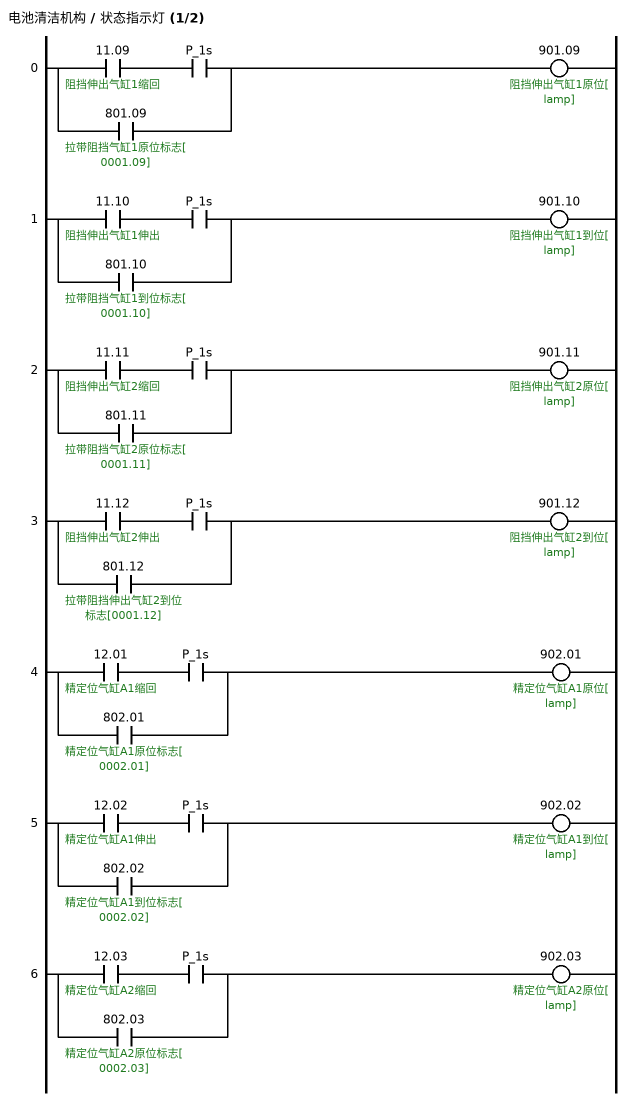
; [picture p72: 电池清洁机构 / 状态指示灯, rungs 0-6]
; rung 0
LD 11.09  ; 阻挡伸出气缸1缩回
AND P_1s
OR 801.09  ; 拉带阻挡气缸1原位标志[0001.09]
OUT 901.09  ; 阻挡伸出气缸1原位[lamp]
; rung 1
LD 11.10  ; 阻挡伸出气缸1伸出
AND P_1s
OR 801.10  ; 拉带阻挡气缸1到位标志[0001.10]
OUT 901.10  ; 阻挡伸出气缸1到位[lamp]
; rung 2
LD 11.11  ; 阻挡伸出气缸2缩回
AND P_1s
OR 801.11  ; 拉带阻挡气缸2原位标志[0001.11]
OUT 901.11  ; 阻挡伸出气缸2原位[lamp]
; rung 3
LD 11.12  ; 阻挡伸出气缸2伸出
AND P_1s
OR 801.12  ; 拉带阻挡伸出气缸2到位标志[0001.12]
OUT 901.12  ; 阻挡伸出气缸2到位[lamp]
; rung 4
LD 12.01  ; 精定位气缸A1缩回
AND P_1s
OR 802.01  ; 精定位气缸A1原位标志[0002.01]
OUT 902.01  ; 精定位气缸A1原位[lamp]
; rung 5
LD 12.02  ; 精定位气缸A1伸出
AND P_1s
OR 802.02  ; 精定位气缸A1到位标志[0002.02]
OUT 902.02  ; 精定位气缸A1到位[lamp]
; rung 6
LD 12.03  ; 精定位气缸A2缩回
AND P_1s
OR 802.03  ; 精定位气缸A2原位标志[0002.03]
OUT 902.03  ; 精定位气缸A2原位[lamp]

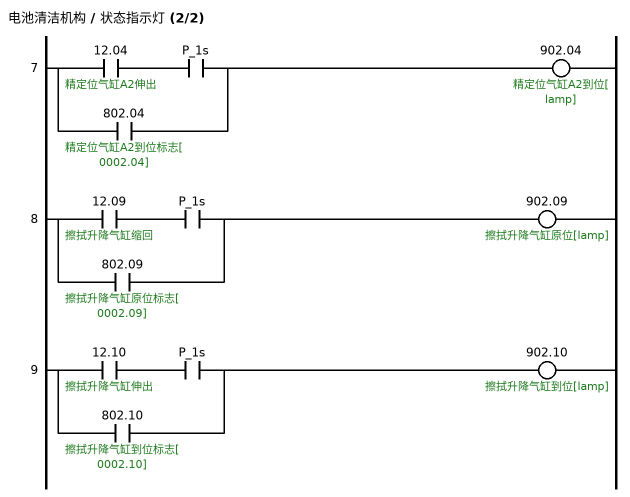
; rung 7
LD 12.04  ; 精定位气缸A2伸出
AND P_1s
OR 802.04  ; 精定位气缸A2到位标志[0002.04]
OUT 902.04  ; 精定位气缸A2到位[lamp]
; rung 8
LD 12.09  ; 擦拭升降气缸缩回
AND P_1s
OR 802.09  ; 擦拭升降气缸原位标志[0002.09]
OUT 902.09  ; 擦拭升降气缸原位[lamp]
; rung 9
LD 12.10  ; 擦拭升降气缸伸出
AND P_1s
OR 802.10  ; 擦拭升降气缸到位标志[0002.10]
OUT 902.10  ; 擦拭升降气缸到位[lamp]

### Section 输出程序

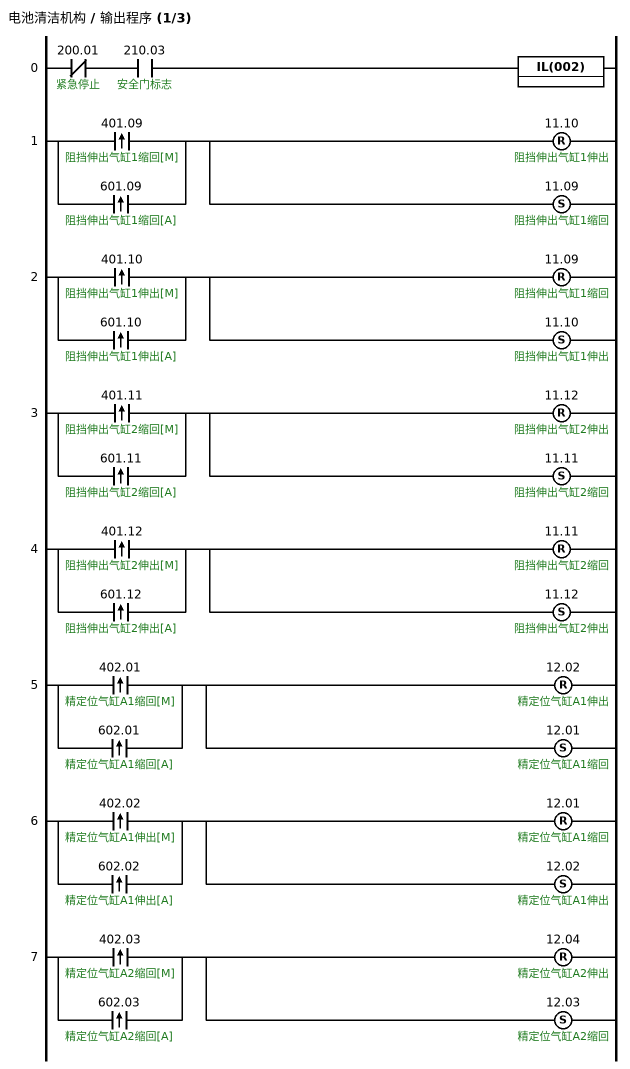
; rung 0
LDNOT 200.01  ; 紧急停止
AND 210.03  ; 安全门标志
IL(002)
; rung 1
@LD 401.09  ; 阻挡伸出气缸1缩回[M]
@OR 601.09  ; 阻挡伸出气缸1缩回[A]
RSET 11.10  ; 阻挡伸出气缸1伸出
SET 11.09  ; 阻挡伸出气缸1缩回
; rung 2
@LD 401.10  ; 阻挡伸出气缸1伸出[M]
@OR 601.10  ; 阻挡伸出气缸1伸出[A]
RSET 11.09  ; 阻挡伸出气缸1缩回
SET 11.10  ; 阻挡伸出气缸1伸出
; rung 3
@LD 401.11  ; 阻挡伸出气缸2缩回[M]
@OR 601.11  ; 阻挡伸出气缸2缩回[A]
RSET 11.12  ; 阻挡伸出气缸2伸出
SET 11.11  ; 阻挡伸出气缸2缩回
; rung 4
@LD 401.12  ; 阻挡伸出气缸2伸出[M]
@OR 601.12  ; 阻挡伸出气缸2伸出[A]
RSET 11.11  ; 阻挡伸出气缸2缩回
SET 11.12  ; 阻挡伸出气缸2伸出
; rung 5
@LD 402.01  ; 精定位气缸A1缩回[M]
@OR 602.01  ; 精定位气缸A1缩回[A]
RSET 12.02  ; 精定位气缸A1伸出
SET 12.01  ; 精定位气缸A1缩回
; rung 6
@LD 402.02  ; 精定位气缸A1伸出[M]
@OR 602.02  ; 精定位气缸A1伸出[A]
RSET 12.01  ; 精定位气缸A1缩回
SET 12.02  ; 精定位气缸A1伸出
; rung 7
@LD 402.03  ; 精定位气缸A2缩回[M]
@OR 602.03  ; 精定位气缸A2缩回[A]
RSET 12.04  ; 精定位气缸A2伸出
SET 12.03  ; 精定位气缸A2缩回

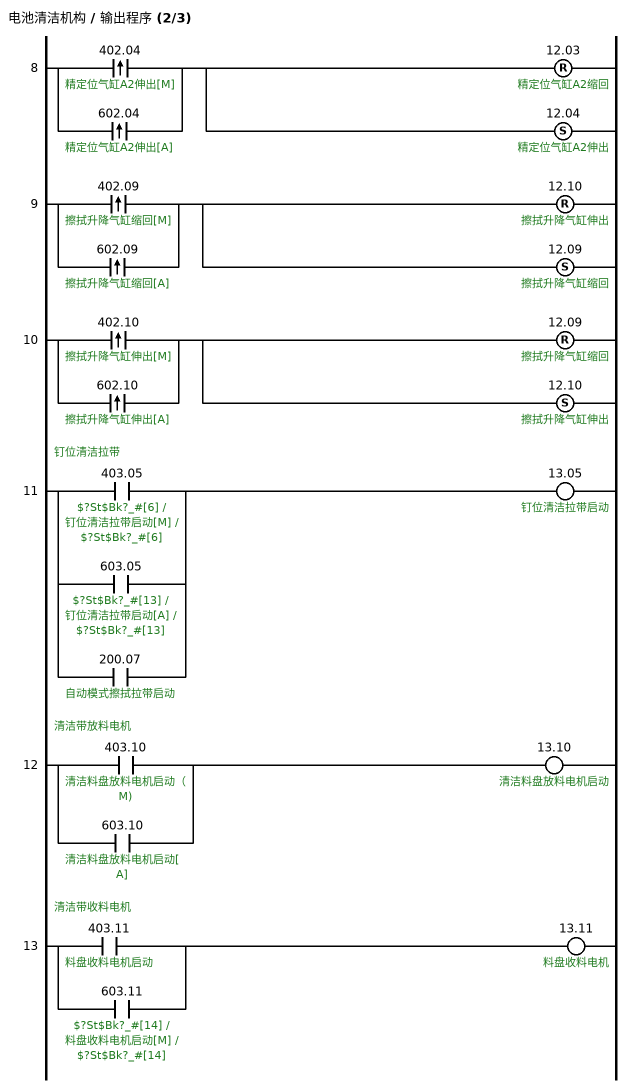
; rung 8
@LD 402.04  ; 精定位气缸A2伸出[M]
@OR 602.04  ; 精定位气缸A2伸出[A]
RSET 12.03  ; 精定位气缸A2缩回
SET 12.04  ; 精定位气缸A2伸出
; rung 9
@LD 402.09  ; 擦拭升降气缸缩回[M]
@OR 602.09  ; 擦拭升降气缸缩回[A]
RSET 12.10  ; 擦拭升降气缸伸出
SET 12.09  ; 擦拭升降气缸缩回
; rung 10
@LD 402.10  ; 擦拭升降气缸伸出[M]
@OR 602.10  ; 擦拭升降气缸伸出[A]
RSET 12.09  ; 擦拭升降气缸缩回
SET 12.10  ; 擦拭升降气缸伸出
; rung 11: 钉位清洁拉带
LD 403.05  ; $?St$Bk?_#[6] / 钉位清洁拉带启动[M] / $?St$Bk?_#[6]
OR 603.05  ; $?St$Bk?_#[13] / 钉位清洁拉带启动[A] / $?St$Bk?_#[13]
OR 200.07  ; 自动模式擦拭拉带启动
OUT 13.05  ; 钉位清洁拉带启动
; rung 12: 清洁带放料电机
LD 403.10  ; 清洁料盘放料电机启动（M)
OR 603.10  ; 清洁料盘放料电机启动[A]
OUT 13.10  ; 清洁料盘放料电机启动
; rung 13: 清洁带收料电机
LD 403.11  ; 料盘收料电机启动
OR 603.11  ; $?St$Bk?_#[14] / 料盘收料电机启动[M] / $?St$Bk?_#[14]
OUT 13.11  ; 料盘收料电机

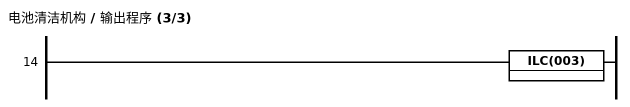
; rung 14
ILC(003)

### Section 擦拭步进电机参数

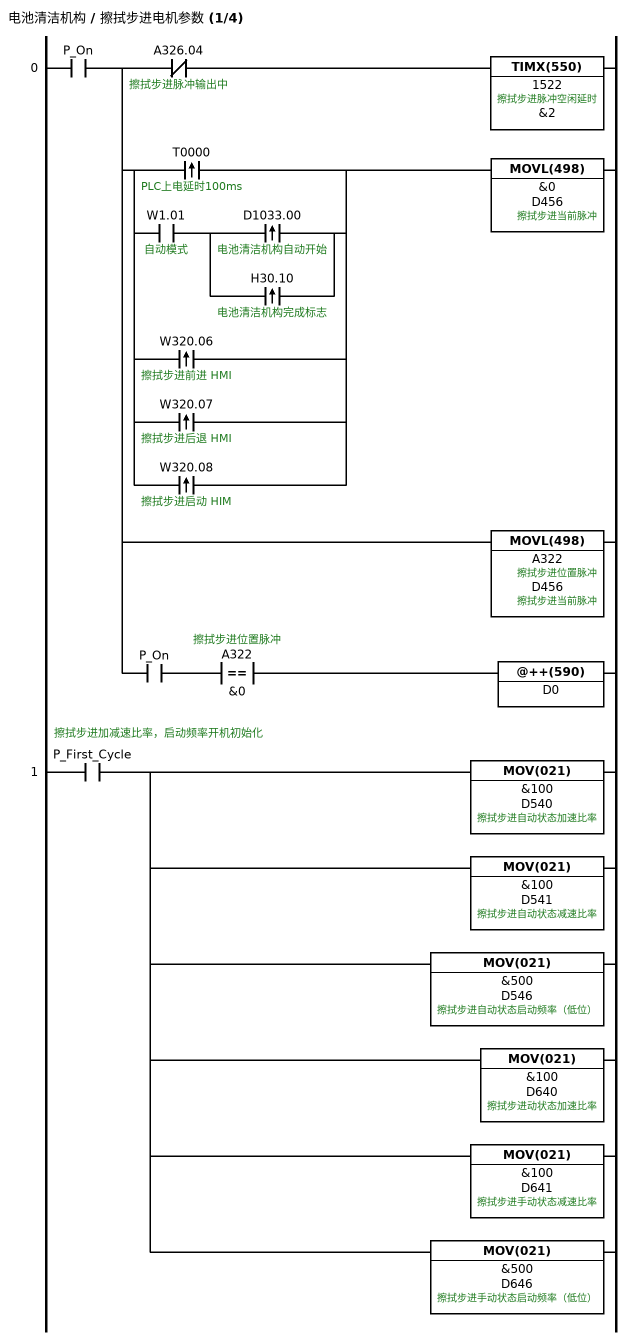
; rung 0
LD P_On
OUT TR0
ANDNOT A326.04  ; 擦拭步进脉冲输出中
TIMX(550) 1522 &2  ; 擦拭步进脉冲空闲延时
LD TR0
@LD T0000  ; PLC上电延时100ms
LD W1.01  ; 自动模式
@LD D1033.00  ; 电池清洁机构自动开始
@OR H30.10  ; 电池清洁机构完成标志
ANDLD
ORLD
@OR W320.06  ; 擦拭步进前进 HMI
@OR W320.07  ; 擦拭步进后退 HMI
@OR W320.08  ; 擦拭步进启动 HIM
ANDLD
MOVL(498) &0 D456  ; 擦拭步进当前脉冲
LD TR0
MOVL(498) A322 D456  ; 擦拭步进位置脉冲, 擦拭步进当前脉冲
AND P_On
AND=L(301) A322 &0  ; 擦拭步进位置脉冲
@++(590) D0
; rung 1: 擦拭步进加减速比率，启动频率开机初始化
LD P_First_Cycle
MOV(021) &100 D540  ; 擦拭步进自动状态加速比率
MOV(021) &100 D541  ; 擦拭步进自动状态减速比率
MOV(021) &500 D546  ; 擦拭步进自动状态启动频率（低位）
MOV(021) &100 D640  ; 擦拭步进动状态加速比率
MOV(021) &100 D641  ; 擦拭步进手动状态减速比率
MOV(021) &500 D646  ; 擦拭步进手动状态启动频率（低位）

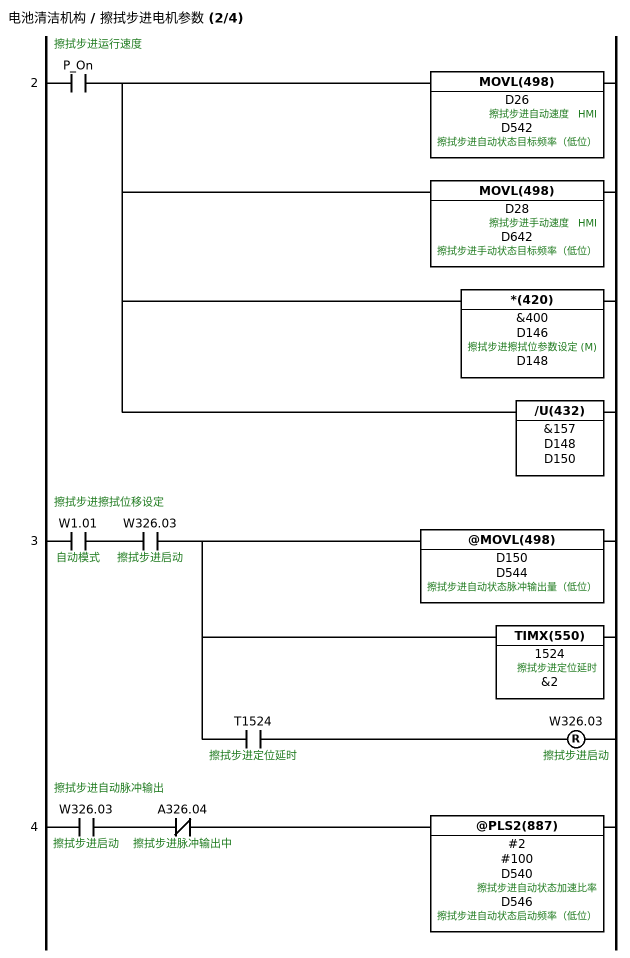
; rung 2: 擦拭步进运行速度
LD P_On
MOVL(498) D26 D542  ; 擦拭步进自动速度   HMI, 擦拭步进自动状态目标频率（低位）
MOVL(498) D28 D642  ; 擦拭步进手动速度   HMI, 擦拭步进手动状态目标频率（低位）
*(420) &400 D146 D148  ; 擦拭步进擦拭位参数设定 (M)
/U(432) &157 D148 D150
; rung 3: 擦拭步进擦拭位移设定
LD W1.01  ; 自动模式
AND W326.03  ; 擦拭步进启动
@MOVL(498) D150 D544  ; 擦拭步进自动状态脉冲输出量（低位）
TIMX(550) 1524 &2  ; 擦拭步进定位延时
AND T1524  ; 擦拭步进定位延时
RSET W326.03  ; 擦拭步进启动
; rung 4: 擦拭步进自动脉冲输出
LD W326.03  ; 擦拭步进启动
ANDNOT A326.04  ; 擦拭步进脉冲输出中
@PLS2(887) #2 #100 D540 D546  ; 擦拭步进自动状态加速比率, 擦拭步进自动状态启动频率（低位）

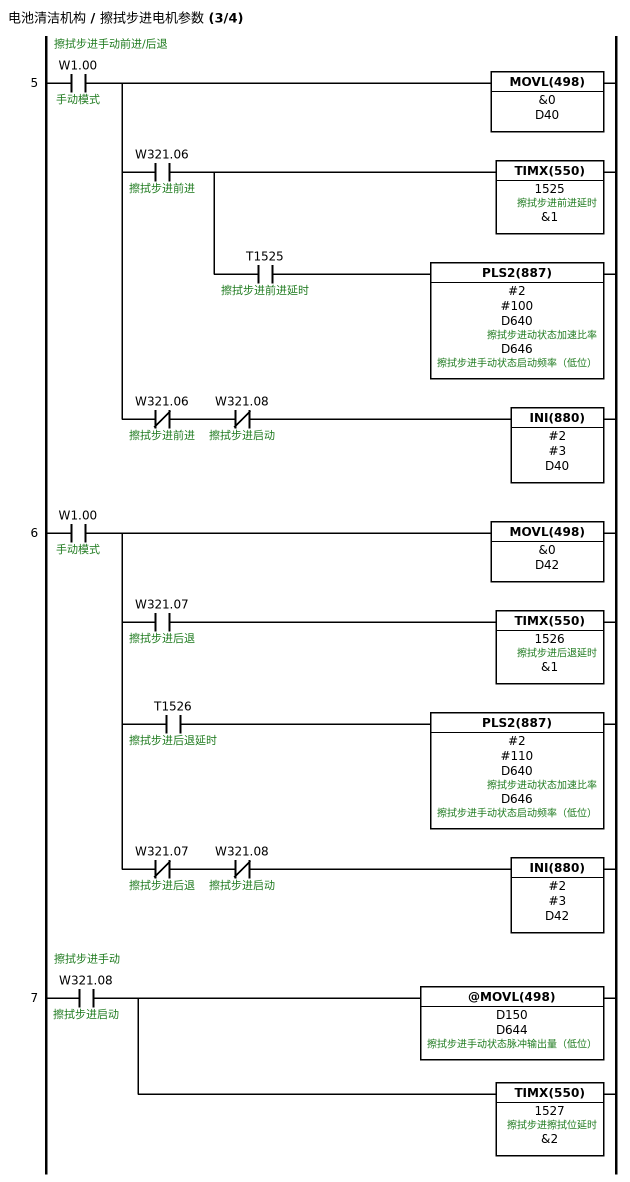
; rung 5: 擦拭步进手动前进/后退
LD W1.00  ; 手动模式
OUT TR0
MOVL(498) &0 D40
AND W321.06  ; 擦拭步进前进
TIMX(550) 1525 &1  ; 擦拭步进前进延时
AND T1525  ; 擦拭步进前进延时
PLS2(887) #2 #100 D640 D646  ; 擦拭步进动状态加速比率, 擦拭步进手动状态启动频率（低位）
LD TR0
ANDNOT W321.06  ; 擦拭步进前进
ANDNOT W321.08  ; 擦拭步进启动
INI(880) #2 #3 D40
; rung 6
LD W1.00  ; 手动模式
OUT TR0
MOVL(498) &0 D42
AND W321.07  ; 擦拭步进后退
TIMX(550) 1526 &1  ; 擦拭步进后退延时
LD TR0
AND T1526  ; 擦拭步进后退延时
PLS2(887) #2 #110 D640 D646  ; 擦拭步进动状态加速比率, 擦拭步进手动状态启动频率（低位）
LD TR0
ANDNOT W321.07  ; 擦拭步进后退
ANDNOT W321.08  ; 擦拭步进启动
INI(880) #2 #3 D42
; rung 7: 擦拭步进手动
LD W321.08  ; 擦拭步进启动
@MOVL(498) D150 D644  ; 擦拭步进手动状态脉冲输出量（低位）
TIMX(550) 1527 &2  ; 擦拭步进擦拭位延时

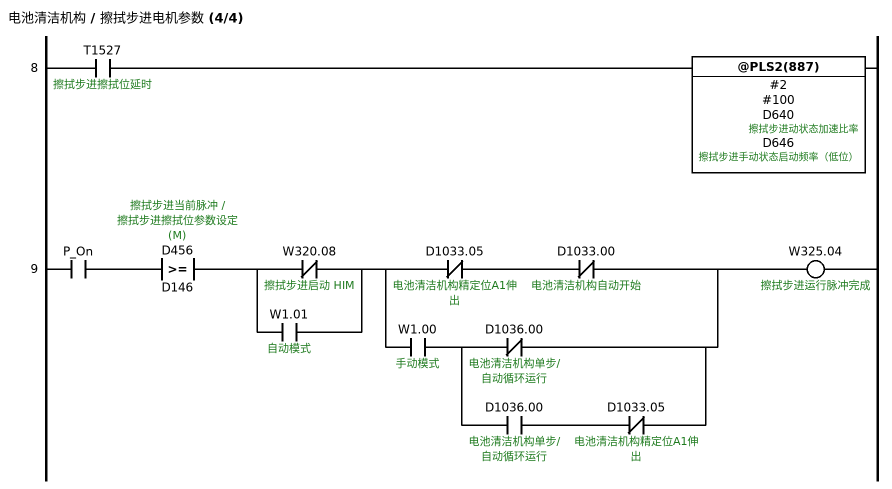
; rung 8
LD T1527  ; 擦拭步进擦拭位延时
@PLS2(887) #2 #100 D640 D646  ; 擦拭步进动状态加速比率, 擦拭步进手动状态启动频率（低位）
; rung 9
LD P_On
AND>=SL(328) D456 D146  ; 擦拭步进当前脉冲, 擦拭步进擦拭位参数设定 (M)
LDNOT W320.08  ; 擦拭步进启动 HIM
OR W1.01  ; 自动模式
ANDLD
LDNOT D1033.05  ; 电池清洁机构精定位A1伸出
ANDNOT D1033.00  ; 电池清洁机构自动开始
LD W1.00  ; 手动模式
LDNOT D1036.00  ; 电池清洁机构单步/自动循环运行
LD D1036.00  ; 电池清洁机构单步/自动循环运行
ANDNOT D1033.05  ; 电池清洁机构精定位A1伸出
ORLD
ANDLD
ORLD
ANDLD
OUT W325.04  ; 擦拭步进运行脉冲完成

### Section END
; rung 0
END(001)

## Program 电池入钉机构 (cyclic task 4)

### Section 主程序

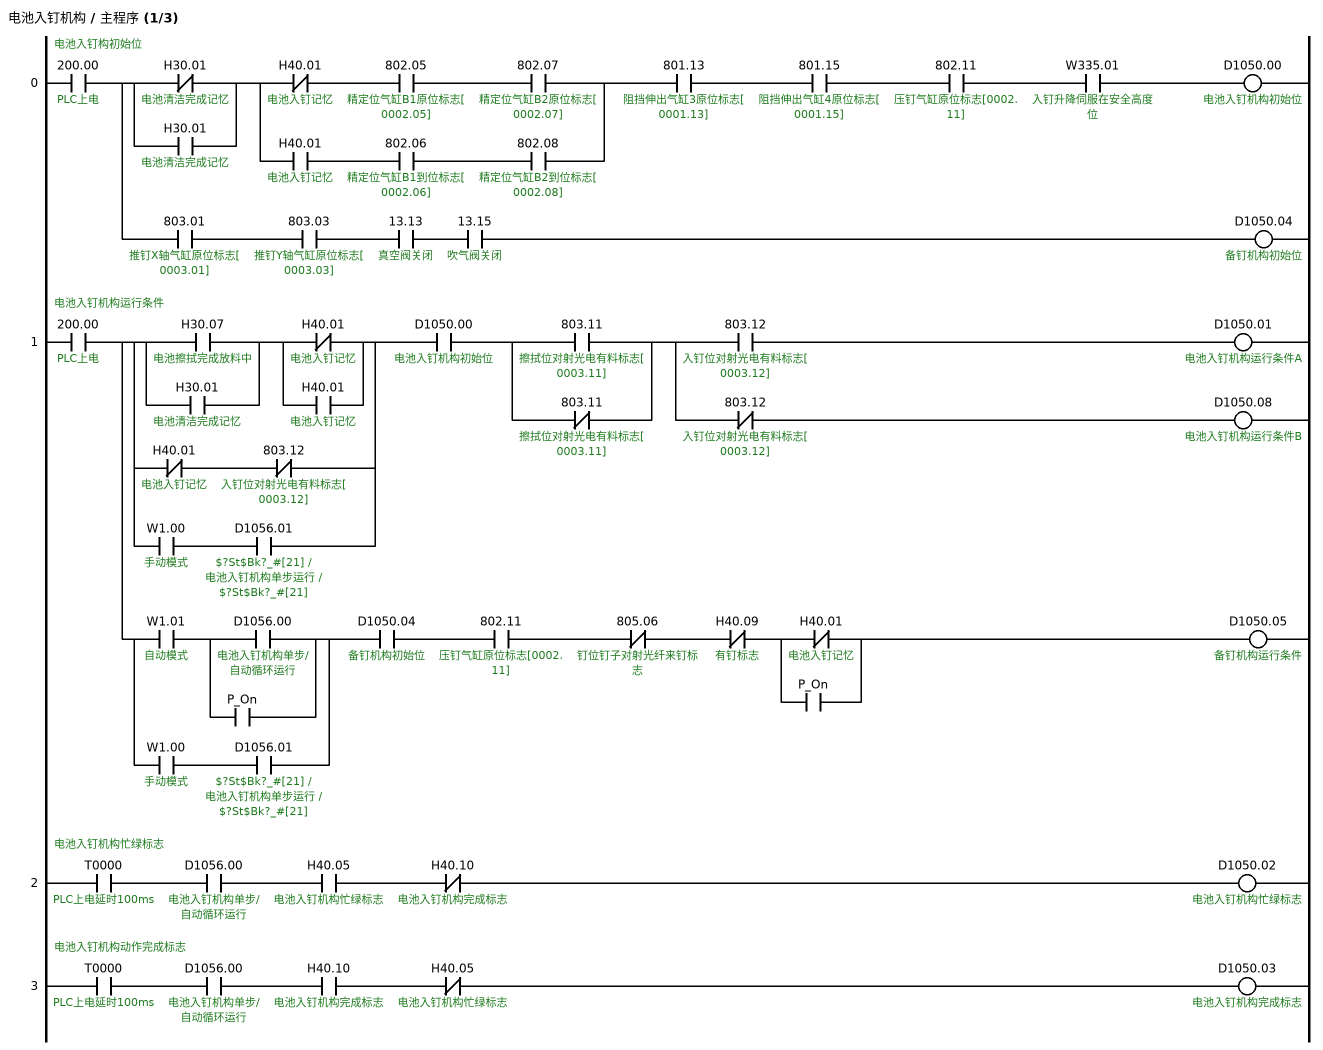
; rung 0: 电池入钉构初始位
LD 200.00  ; PLC上电
OUT TR0
LDNOT H30.01  ; 电池清洁完成记忆
OR H30.01  ; 电池清洁完成记忆
ANDLD
LDNOT H40.01  ; 电池入钉记忆
AND 802.05  ; 精定位气缸B1原位标志[0002.05]
AND 802.07  ; 精定位气缸B2原位标志[0002.07]
LD H40.01  ; 电池入钉记忆
AND 802.06  ; 精定位气缸B1到位标志[0002.06]
AND 802.08  ; 精定位气缸B2到位标志[0002.08]
ORLD
ANDLD
AND 801.13  ; 阻挡伸出气缸3原位标志[0001.13]
AND 801.15  ; 阻挡伸出气缸4原位标志[0001.15]
AND 802.11  ; 压钉气缸原位标志[0002.11]
AND W335.01  ; 入钉升降伺服在安全高度位
OUT D1050.00  ; 电池入钉机构初始位
LD TR0
AND 803.01  ; 推钉X轴气缸原位标志[0003.01]
AND 803.03  ; 推钉Y轴气缸原位标志[0003.03]
AND 13.13  ; 真空阀关闭
AND 13.15  ; 吹气阀关闭
OUT D1050.04  ; 备钉机构初始位
; rung 1: 电池入钉机构运行条件
LD 200.00  ; PLC上电
OUT TR0
LD H30.07  ; 电池擦拭完成放料中
OR H30.01  ; 电池清洁完成记忆
LDNOT H40.01  ; 电池入钉记忆
OR H40.01  ; 电池入钉记忆
ANDLD
LDNOT H40.01  ; 电池入钉记忆
ANDNOT 803.12  ; 入钉位对射光电有料标志[0003.12]
ORLD
LD W1.00  ; 手动模式
AND D1056.01  ; $?St$Bk?_#[21] / 电池入钉机构单步运行 / $?St$Bk?_#[21]
ORLD
ANDLD
AND D1050.00  ; 电池入钉机构初始位
LD 803.11  ; 擦拭位对射光电有料标志[0003.11]
ORNOT 803.11  ; 擦拭位对射光电有料标志[0003.11]
ANDLD
OUT TR1
AND 803.12  ; 入钉位对射光电有料标志[0003.12]
OUT D1050.01  ; 电池入钉机构运行条件A
LD TR1
ANDNOT 803.12  ; 入钉位对射光电有料标志[0003.12]
OUT D1050.08  ; 电池入钉机构运行条件B
LD TR0
LD W1.01  ; 自动模式
LD D1056.00  ; 电池入钉机构单步/自动循环运行
OR P_On
ANDLD
LD W1.00  ; 手动模式
AND D1056.01  ; $?St$Bk?_#[21] / 电池入钉机构单步运行 / $?St$Bk?_#[21]
ORLD
ANDLD
AND D1050.04  ; 备钉机构初始位
AND 802.11  ; 压钉气缸原位标志[0002.11]
ANDNOT 805.06  ; 钉位钉子对射光纤来钉标志
ANDNOT H40.09  ; 有钉标志
LDNOT H40.01  ; 电池入钉记忆
OR P_On
ANDLD
OUT D1050.05  ; 备钉机构运行条件
; rung 2: 电池入钉机构忙绿标志
LD T0000  ; PLC上电延时100ms
AND D1056.00  ; 电池入钉机构单步/自动循环运行
AND H40.05  ; 电池入钉机构忙绿标志
ANDNOT H40.10  ; 电池入钉机构完成标志
OUT D1050.02  ; 电池入钉机构忙绿标志
; rung 3: 电池入钉机构动作完成标志
LD T0000  ; PLC上电延时100ms
AND D1056.00  ; 电池入钉机构单步/自动循环运行
AND H40.10  ; 电池入钉机构完成标志
ANDNOT H40.05  ; 电池入钉机构忙绿标志
OUT D1050.03  ; 电池入钉机构完成标志

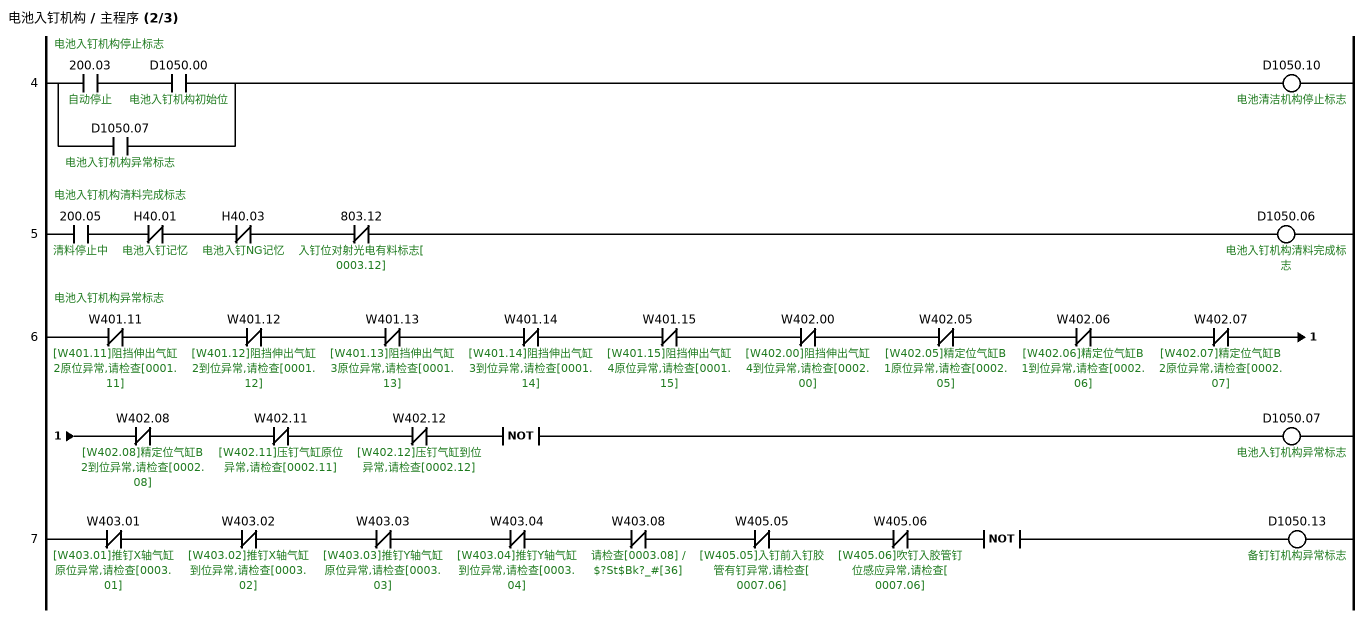
; rung 4: 电池入钉机构停止标志
LD 200.03  ; 自动停止
AND D1050.00  ; 电池入钉机构初始位
OR D1050.07  ; 电池入钉机构异常标志
OUT D1050.10  ; 电池清洁机构停止标志
; rung 5: 电池入钉机构清料完成标志
LD 200.05  ; 清料停止中
ANDNOT H40.01  ; 电池入钉记忆
ANDNOT H40.03  ; 电池入钉NG记忆
ANDNOT 803.12  ; 入钉位对射光电有料标志[0003.12]
OUT D1050.06  ; 电池入钉机构清料完成标志
; rung 6: 电池入钉机构异常标志
LDNOT W401.11  ; [W401.11]阻挡伸出气缸2原位异常,请检查[0001.11]
ANDNOT W401.12  ; [W401.12]阻挡伸出气缸2到位异常,请检查[0001.12]
ANDNOT W401.13  ; [W401.13]阻挡伸出气缸3原位异常,请检查[0001.13]
ANDNOT W401.14  ; [W401.14]阻挡伸出气缸3到位异常,请检查[0001.14]
ANDNOT W401.15  ; [W401.15]阻挡伸出气缸4原位异常,请检查[0001.15]
ANDNOT W402.00  ; [W402.00]阻挡伸出气缸4到位异常,请检查[0002.00]
ANDNOT W402.05  ; [W402.05]精定位气缸B1原位异常,请检查[0002.05]
ANDNOT W402.06  ; [W402.06]精定位气缸B1到位异常,请检查[0002.06]
ANDNOT W402.07  ; [W402.07]精定位气缸B2原位异常,请检查[0002.07]
ANDNOT W402.08  ; [W402.08]精定位气缸B2到位异常,请检查[0002.08]
ANDNOT W402.11  ; [W402.11]压钉气缸原位异常,请检查[0002.11]
ANDNOT W402.12  ; [W402.12]压钉气缸到位异常,请检查[0002.12]
NOT(520)
OUT D1050.07  ; 电池入钉机构异常标志
; rung 7
LDNOT W403.01  ; [W403.01]推钉X轴气缸原位异常,请检查[0003.01]
ANDNOT W403.02  ; [W403.02]推钉X轴气缸到位异常,请检查[0003.02]
ANDNOT W403.03  ; [W403.03]推钉Y轴气缸原位异常,请检查[0003.03]
ANDNOT W403.04  ; [W403.04]推钉Y轴气缸到位异常,请检查[0003.04]
ANDNOT W403.08  ; 请检查[0003.08] / $?St$Bk?_#[36]
ANDNOT W405.05  ; [W405.05]入钉前入钉胶管有钉异常,请检查[0007.06]
ANDNOT W405.06  ; [W405.06]吹钉入胶管钉位感应异常,请检查[0007.06]
NOT(520)
OUT D1050.13  ; 备钉钉机构异常标志

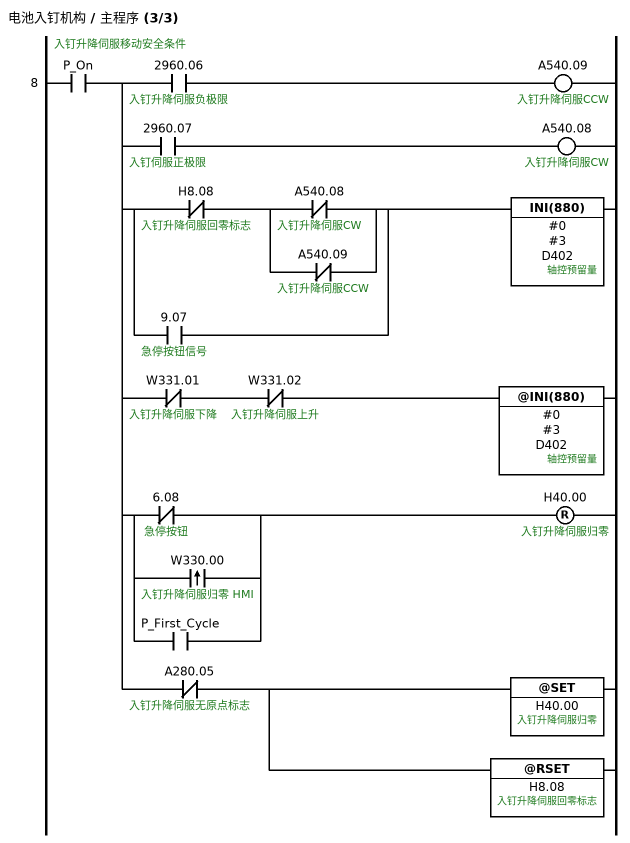
; rung 8: 入钉升降伺服移动安全条件
LD P_On
OUT TR0
AND 2960.06  ; 入钉升降伺服负极限
OUT A540.09  ; 入钉升降伺服CCW
LD TR0
AND 2960.07  ; 入钉伺服正极限
OUT A540.08  ; 入钉升降伺服CW
LD TR0
LDNOT H8.08  ; 入钉升降伺服回零标志
LDNOT A540.08  ; 入钉升降伺服CW
ORNOT A540.09  ; 入钉升降伺服CCW
ANDLD
OR 9.07  ; 急停按钮信号
ANDLD
INI(880) #0 #3 D402  ; 轴控预留量
LD TR0
ANDNOT W331.01  ; 入钉升降伺服下降
ANDNOT W331.02  ; 入钉升降伺服上升
@INI(880) #0 #3 D402  ; 轴控预留量
LD TR0
LDNOT 6.08  ; 急停按钮
@OR W330.00  ; 入钉升降伺服归零 HMI
OR P_First_Cycle
ANDLD
RSET H40.00  ; 入钉升降伺服归零
LD TR0
ANDNOT A280.05  ; 入钉升降伺服无原点标志
@SET H40.00  ; 入钉升降伺服归零
@RSET H8.08  ; 入钉升降伺服回零标志

### Section 工站复位

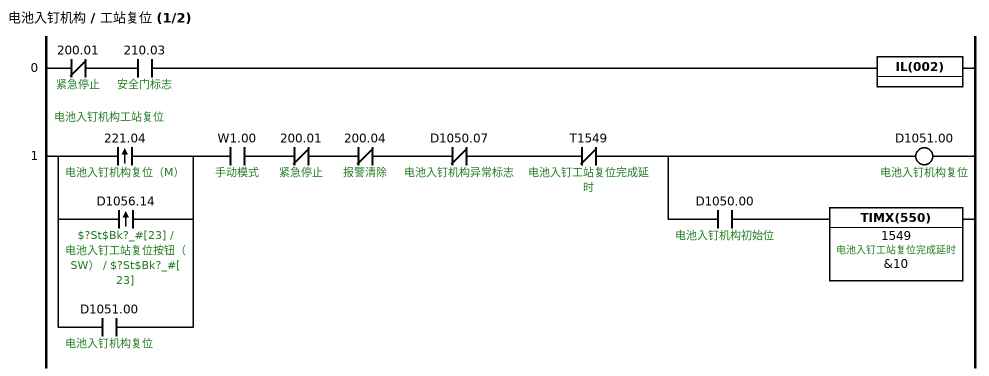
; rung 0
LDNOT 200.01  ; 紧急停止
AND 210.03  ; 安全门标志
IL(002)
; rung 1: 电池入钉机构工站复位
@LD 221.04  ; 电池入钉机构复位（M）
@OR D1056.14  ; $?St$Bk?_#[23] / 电池入钉工站复位按钮（SW） / $?St$Bk?_#[23]
OR D1051.00  ; 电池入钉机构复位
AND W1.00  ; 手动模式
ANDNOT 200.01  ; 紧急停止
ANDNOT 200.04  ; 报警清除
ANDNOT D1050.07  ; 电池入钉机构异常标志
ANDNOT T1549  ; 电池入钉工站复位完成延时
OUT D1051.00  ; 电池入钉机构复位
AND D1050.00  ; 电池入钉机构初始位
TIMX(550) 1549 &10  ; 电池入钉工站复位完成延时

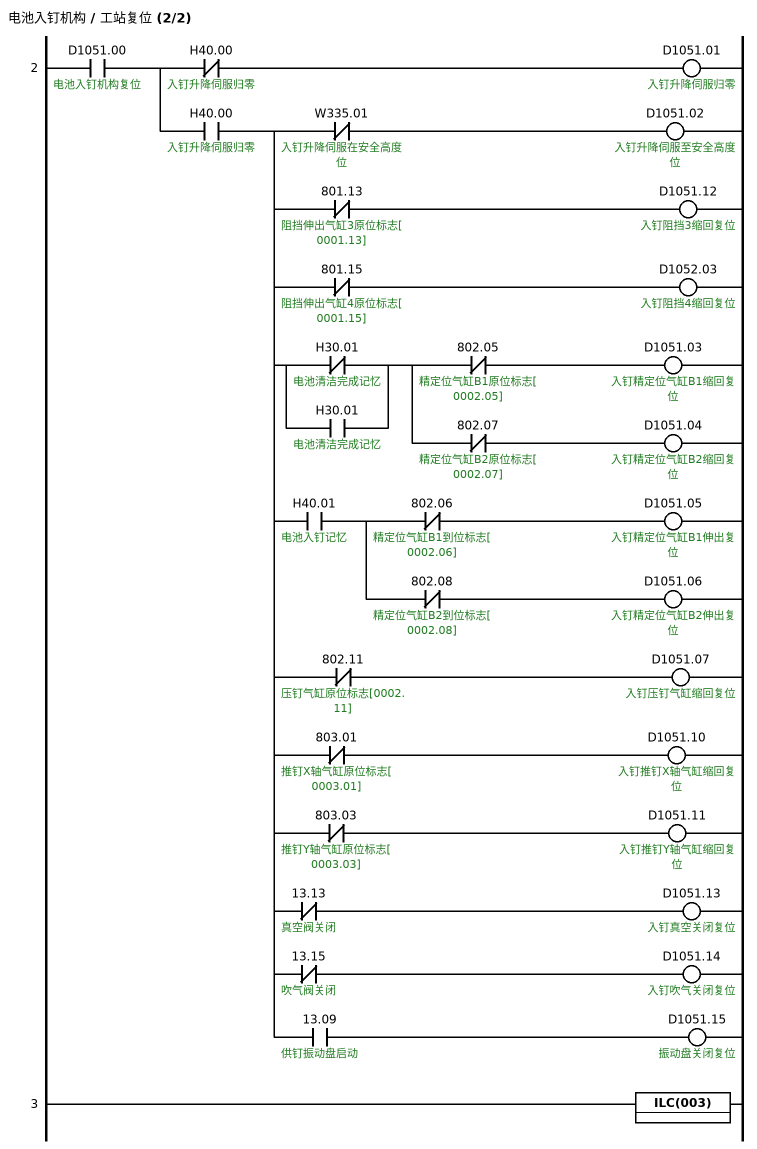
; rung 2
LD D1051.00  ; 电池入钉机构复位
OUT TR0
ANDNOT H40.00  ; 入钉升降伺服归零
OUT D1051.01  ; 入钉升降伺服归零
LD TR0
AND H40.00  ; 入钉升降伺服归零
OUT TR0
ANDNOT W335.01  ; 入钉升降伺服在安全高度位
OUT D1051.02  ; 入钉升降伺服至安全高度位
LD TR0
ANDNOT 801.13  ; 阻挡伸出气缸3原位标志[0001.13]
OUT D1051.12  ; 入钉阻挡3缩回复位
LD TR0
ANDNOT 801.15  ; 阻挡伸出气缸4原位标志[0001.15]
OUT D1052.03  ; 入钉阻挡4缩回复位
LD TR0
LDNOT H30.01  ; 电池清洁完成记忆
OR H30.01  ; 电池清洁完成记忆
ANDLD
OUT TR1
ANDNOT 802.05  ; 精定位气缸B1原位标志[0002.05]
OUT D1051.03  ; 入钉精定位气缸B1缩回复位
LD TR1
ANDNOT 802.07  ; 精定位气缸B2原位标志[0002.07]
OUT D1051.04  ; 入钉精定位气缸B2缩回复位
LD TR0
AND H40.01  ; 电池入钉记忆
OUT TR1
ANDNOT 802.06  ; 精定位气缸B1到位标志[0002.06]
OUT D1051.05  ; 入钉精定位气缸B1伸出复位
LD TR1
ANDNOT 802.08  ; 精定位气缸B2到位标志[0002.08]
OUT D1051.06  ; 入钉精定位气缸B2伸出复位
LD TR0
ANDNOT 802.11  ; 压钉气缸原位标志[0002.11]
OUT D1051.07  ; 入钉压钉气缸缩回复位
LD TR0
ANDNOT 803.01  ; 推钉X轴气缸原位标志[0003.01]
OUT D1051.10  ; 入钉推钉X轴气缸缩回复位
LD TR0
ANDNOT 803.03  ; 推钉Y轴气缸原位标志[0003.03]
OUT D1051.11  ; 入钉推钉Y轴气缸缩回复位
LD TR0
ANDNOT 13.13  ; 真空阀关闭
OUT D1051.13  ; 入钉真空关闭复位
LD TR0
ANDNOT 13.15  ; 吹气阀关闭
OUT D1051.14  ; 入钉吹气关闭复位
LD TR0
AND 13.09  ; 供钉振动盘启动
OUT D1051.15  ; 振动盘关闭复位
; rung 3
ILC(003)

### Section 手动程序

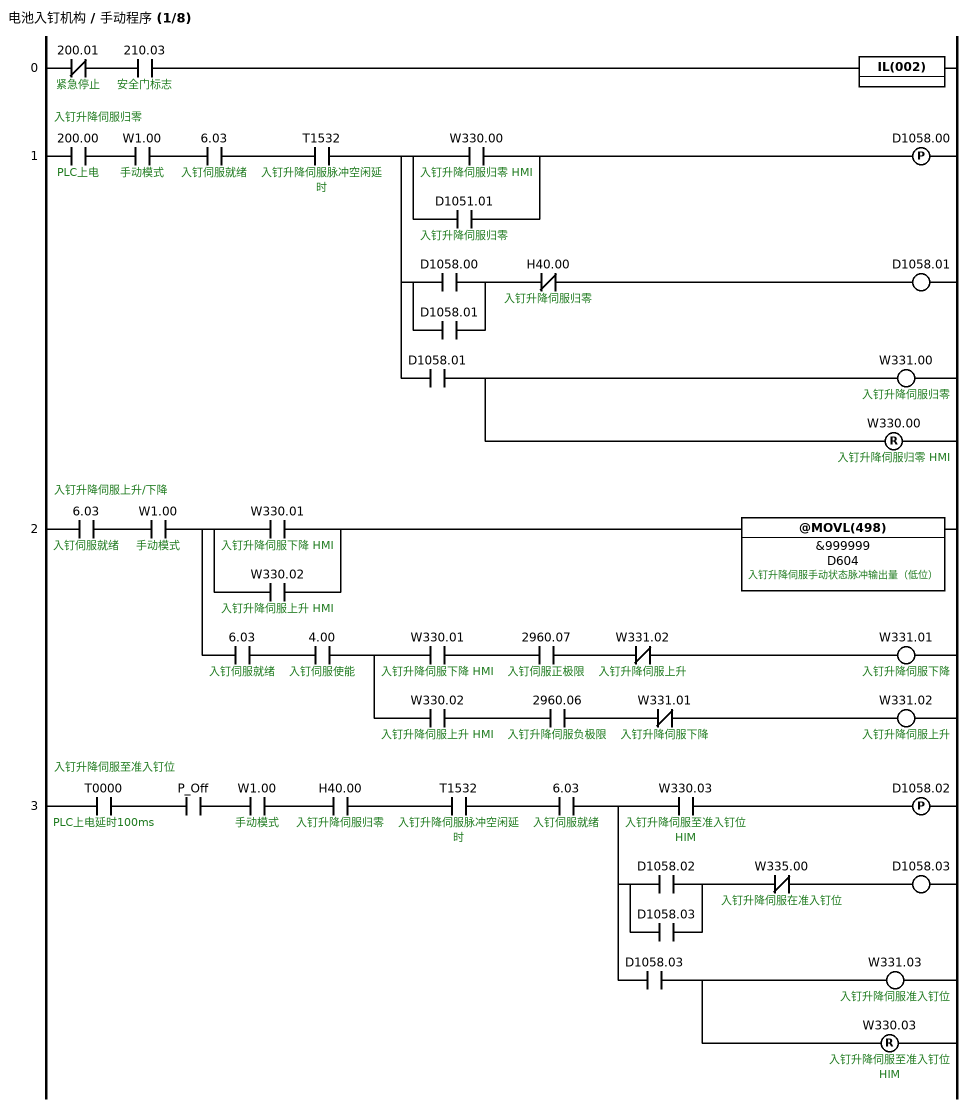
; rung 0
LDNOT 200.01  ; 紧急停止
AND 210.03  ; 安全门标志
IL(002)
; rung 1: 入钉升降伺服归零
LD 200.00  ; PLC上电
AND W1.00  ; 手动模式
AND 6.03  ; 入钉伺服就绪
AND T1532  ; 入钉升降伺服脉冲空闲延时
OUT TR0
LD W330.00  ; 入钉升降伺服归零 HMI
OR D1051.01  ; 入钉升降伺服归零
ANDLD
DIFU(013) D1058.00
LD TR0
LD D1058.00
OR D1058.01
ANDLD
ANDNOT H40.00  ; 入钉升降伺服归零
OUT D1058.01
LD TR0
AND D1058.01
OUT W331.00  ; 入钉升降伺服归零
RSET W330.00  ; 入钉升降伺服归零 HMI
; rung 2: 入钉升降伺服上升/下降
LD 6.03  ; 入钉伺服就绪
AND W1.00  ; 手动模式
OUT TR0
LD W330.01  ; 入钉升降伺服下降 HMI
OR W330.02  ; 入钉升降伺服上升 HMI
ANDLD
@MOVL(498) &999999 D604  ; 入钉升降伺服手动状态脉冲输出量（低位）
LD TR0
AND 6.03  ; 入钉伺服就绪
AND 4.00  ; 入钉伺服使能
OUT TR0
AND W330.01  ; 入钉升降伺服下降 HMI
AND 2960.07  ; 入钉伺服正极限
ANDNOT W331.02  ; 入钉升降伺服上升
OUT W331.01  ; 入钉升降伺服下降
LD TR0
AND W330.02  ; 入钉升降伺服上升 HMI
AND 2960.06  ; 入钉升降伺服负极限
ANDNOT W331.01  ; 入钉升降伺服下降
OUT W331.02  ; 入钉升降伺服上升
; rung 3: 入钉升降伺服至准入钉位
LD T0000  ; PLC上电延时100ms
AND P_Off
AND W1.00  ; 手动模式
AND H40.00  ; 入钉升降伺服归零
AND T1532  ; 入钉升降伺服脉冲空闲延时
AND 6.03  ; 入钉伺服就绪
OUT TR0
AND W330.03  ; 入钉升降伺服至准入钉位 HIM
DIFU(013) D1058.02
LD TR0
LD D1058.02
OR D1058.03
ANDLD
ANDNOT W335.00  ; 入钉升降伺服在准入钉位
OUT D1058.03
LD TR0
AND D1058.03
OUT W331.03  ; 入钉升降伺服准入钉位
RSET W330.03  ; 入钉升降伺服至准入钉位 HIM

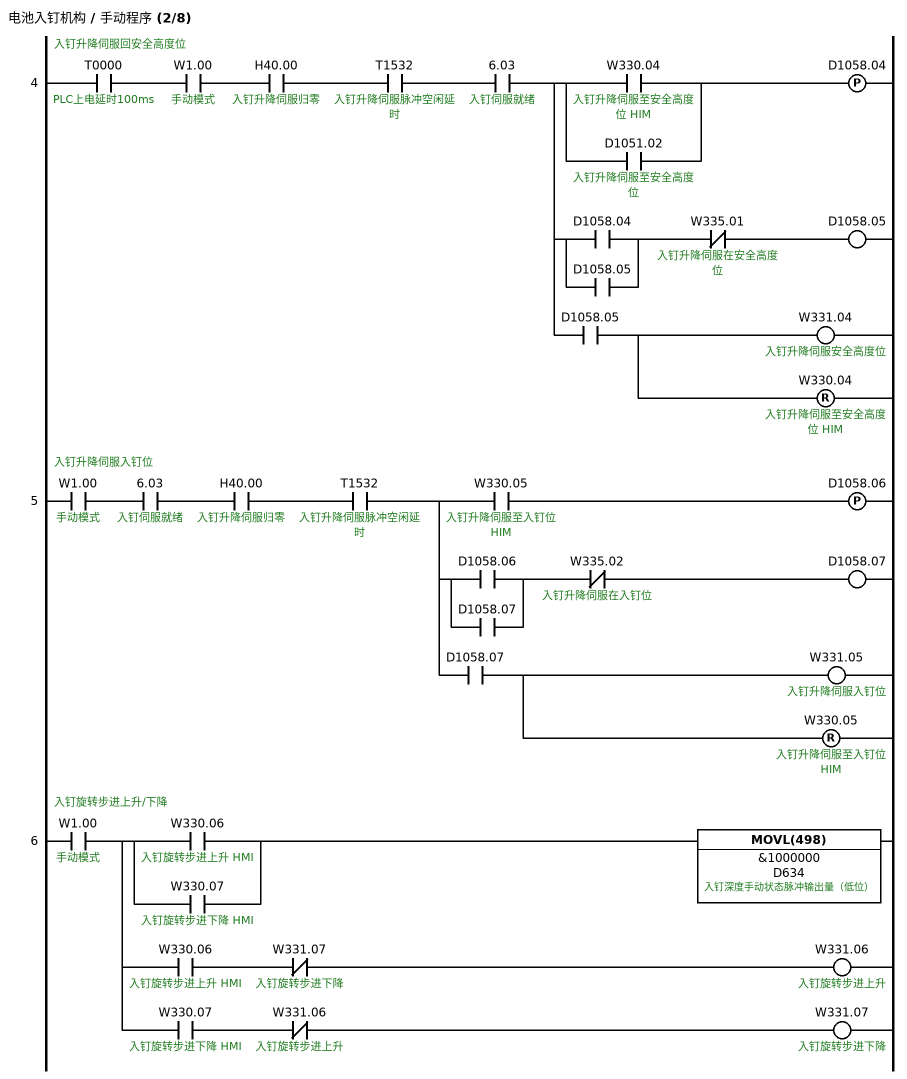
; rung 4: 入钉升降伺服回安全高度位
LD T0000  ; PLC上电延时100ms
AND W1.00  ; 手动模式
AND H40.00  ; 入钉升降伺服归零
AND T1532  ; 入钉升降伺服脉冲空闲延时
AND 6.03  ; 入钉伺服就绪
OUT TR0
LD W330.04  ; 入钉升降伺服至安全高度位 HIM
OR D1051.02  ; 入钉升降伺服至安全高度位
ANDLD
DIFU(013) D1058.04
LD TR0
LD D1058.04
OR D1058.05
ANDLD
ANDNOT W335.01  ; 入钉升降伺服在安全高度位
OUT D1058.05
LD TR0
AND D1058.05
OUT W331.04  ; 入钉升降伺服安全高度位
RSET W330.04  ; 入钉升降伺服至安全高度位 HIM
; rung 5: 入钉升降伺服入钉位
LD W1.00  ; 手动模式
AND 6.03  ; 入钉伺服就绪
AND H40.00  ; 入钉升降伺服归零
AND T1532  ; 入钉升降伺服脉冲空闲延时
OUT TR0
AND W330.05  ; 入钉升降伺服至入钉位 HIM
DIFU(013) D1058.06
LD TR0
LD D1058.06
OR D1058.07
ANDLD
ANDNOT W335.02  ; 入钉升降伺服在入钉位
OUT D1058.07
LD TR0
AND D1058.07
OUT W331.05  ; 入钉升降伺服入钉位
RSET W330.05  ; 入钉升降伺服至入钉位 HIM
; rung 6: 入钉旋转步进上升/下降
LD W1.00  ; 手动模式
OUT TR0
LD W330.06  ; 入钉旋转步进上升 HMI
OR W330.07  ; 入钉旋转步进下降 HMI
ANDLD
MOVL(498) &1000000 D634  ; 入钉深度手动状态脉冲输出量（低位）
LD TR0
AND W330.06  ; 入钉旋转步进上升 HMI
ANDNOT W331.07  ; 入钉旋转步进下降
OUT W331.06  ; 入钉旋转步进上升
LD TR0
AND W330.07  ; 入钉旋转步进下降 HMI
ANDNOT W331.06  ; 入钉旋转步进上升
OUT W331.07  ; 入钉旋转步进下降

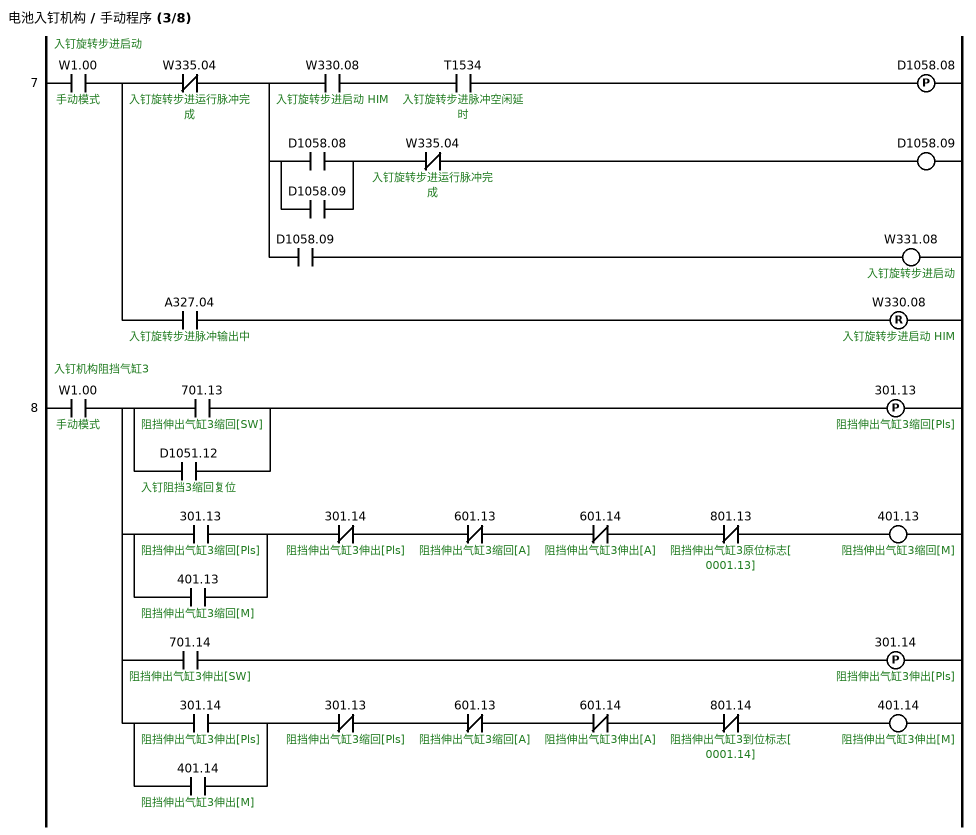
; rung 7: 入钉旋转步进启动
LD W1.00  ; 手动模式
OUT TR0
ANDNOT W335.04  ; 入钉旋转步进运行脉冲完成
OUT TR1
AND W330.08  ; 入钉旋转步进启动 HIM
AND T1534  ; 入钉旋转步进脉冲空闲延时
DIFU(013) D1058.08
LD TR1
LD D1058.08
OR D1058.09
ANDLD
ANDNOT W335.04  ; 入钉旋转步进运行脉冲完成
OUT D1058.09
LD TR1
AND D1058.09
OUT W331.08  ; 入钉旋转步进启动
LD TR0
AND A327.04  ; 入钉旋转步进脉冲输出中
RSET W330.08  ; 入钉旋转步进启动 HIM
; rung 8: 入钉机构阻挡气缸3
LD W1.00  ; 手动模式
OUT TR0
LD 701.13  ; 阻挡伸出气缸3缩回[SW]
OR D1051.12  ; 入钉阻挡3缩回复位
ANDLD
DIFU(013) 301.13  ; 阻挡伸出气缸3缩回[Pls]
LD TR0
LD 301.13  ; 阻挡伸出气缸3缩回[Pls]
OR 401.13  ; 阻挡伸出气缸3缩回[M]
ANDLD
ANDNOT 301.14  ; 阻挡伸出气缸3伸出[Pls]
ANDNOT 601.13  ; 阻挡伸出气缸3缩回[A]
ANDNOT 601.14  ; 阻挡伸出气缸3伸出[A]
ANDNOT 801.13  ; 阻挡伸出气缸3原位标志[0001.13]
OUT 401.13  ; 阻挡伸出气缸3缩回[M]
LD TR0
AND 701.14  ; 阻挡伸出气缸3伸出[SW]
DIFU(013) 301.14  ; 阻挡伸出气缸3伸出[Pls]
LD TR0
LD 301.14  ; 阻挡伸出气缸3伸出[Pls]
OR 401.14  ; 阻挡伸出气缸3伸出[M]
ANDLD
ANDNOT 301.13  ; 阻挡伸出气缸3缩回[Pls]
ANDNOT 601.13  ; 阻挡伸出气缸3缩回[A]
ANDNOT 601.14  ; 阻挡伸出气缸3伸出[A]
ANDNOT 801.14  ; 阻挡伸出气缸3到位标志[0001.14]
OUT 401.14  ; 阻挡伸出气缸3伸出[M]

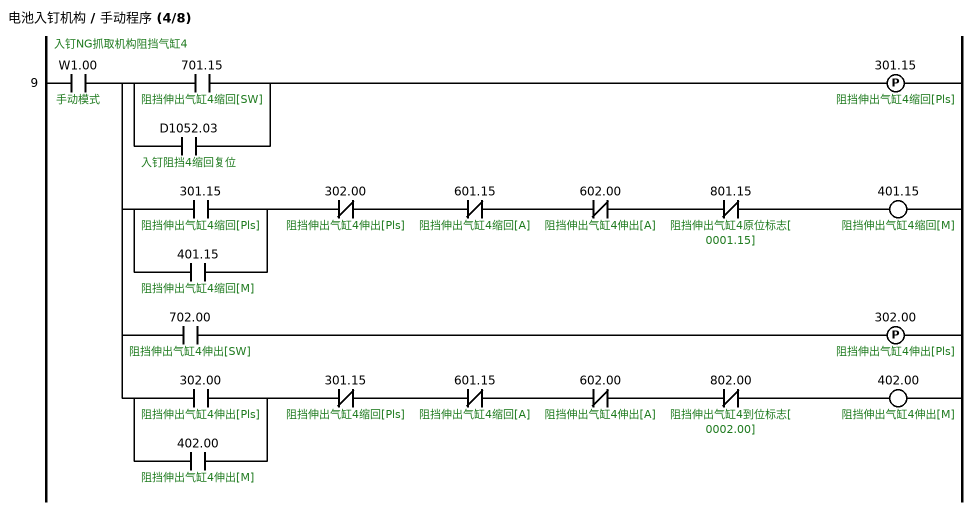
; rung 9: 入钉NG抓取机构阻挡气缸4
LD W1.00  ; 手动模式
OUT TR0
LD 701.15  ; 阻挡伸出气缸4缩回[SW]
OR D1052.03  ; 入钉阻挡4缩回复位
ANDLD
DIFU(013) 301.15  ; 阻挡伸出气缸4缩回[Pls]
LD TR0
LD 301.15  ; 阻挡伸出气缸4缩回[Pls]
OR 401.15  ; 阻挡伸出气缸4缩回[M]
ANDLD
ANDNOT 302.00  ; 阻挡伸出气缸4伸出[Pls]
ANDNOT 601.15  ; 阻挡伸出气缸4缩回[A]
ANDNOT 602.00  ; 阻挡伸出气缸4伸出[A]
ANDNOT 801.15  ; 阻挡伸出气缸4原位标志[0001.15]
OUT 401.15  ; 阻挡伸出气缸4缩回[M]
LD TR0
AND 702.00  ; 阻挡伸出气缸4伸出[SW]
DIFU(013) 302.00  ; 阻挡伸出气缸4伸出[Pls]
LD TR0
LD 302.00  ; 阻挡伸出气缸4伸出[Pls]
OR 402.00  ; 阻挡伸出气缸4伸出[M]
ANDLD
ANDNOT 301.15  ; 阻挡伸出气缸4缩回[Pls]
ANDNOT 601.15  ; 阻挡伸出气缸4缩回[A]
ANDNOT 602.00  ; 阻挡伸出气缸4伸出[A]
ANDNOT 802.00  ; 阻挡伸出气缸4到位标志[0002.00]
OUT 402.00  ; 阻挡伸出气缸4伸出[M]

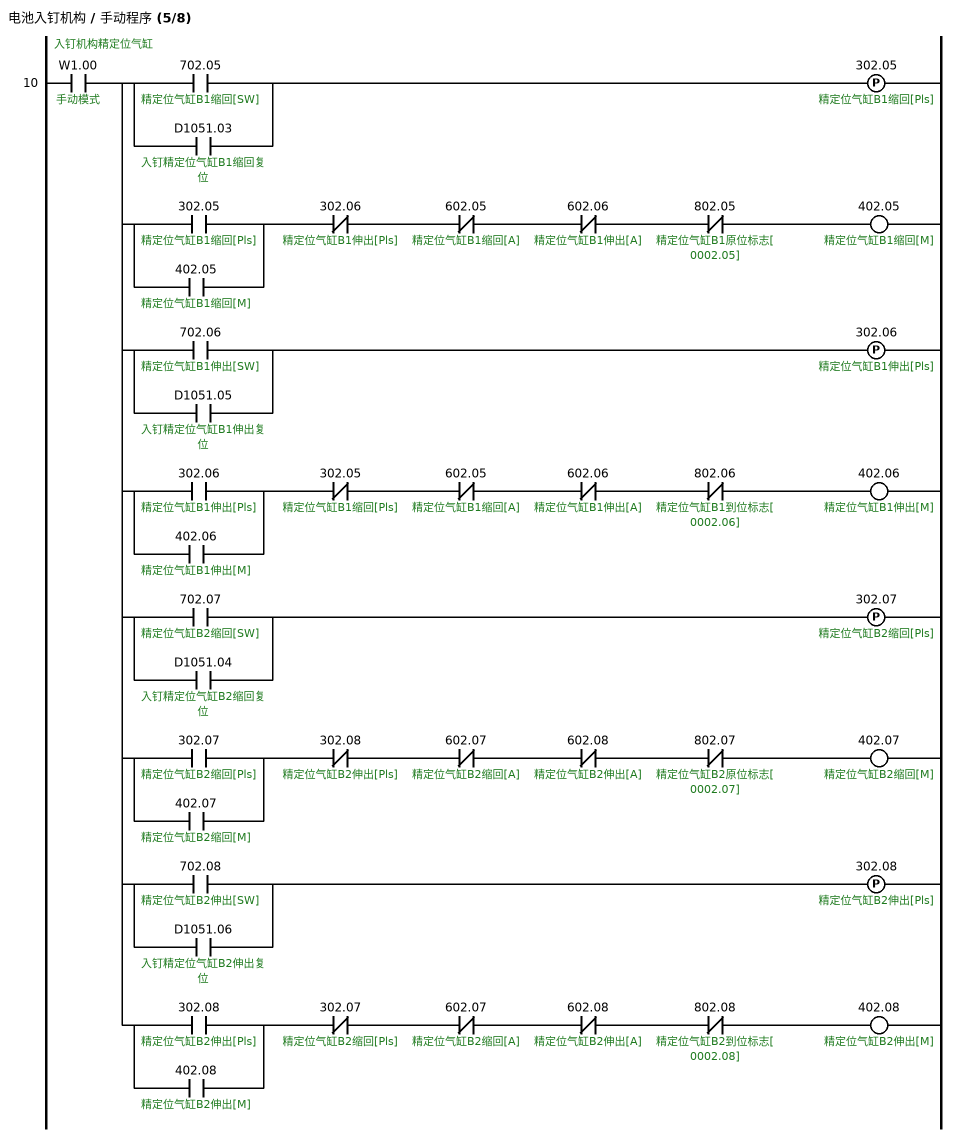
; rung 10: 入钉机构精定位气缸
LD W1.00  ; 手动模式
OUT TR0
LD 702.05  ; 精定位气缸B1缩回[SW]
OR D1051.03  ; 入钉精定位气缸B1缩回复位
ANDLD
DIFU(013) 302.05  ; 精定位气缸B1缩回[Pls]
LD TR0
LD 302.05  ; 精定位气缸B1缩回[Pls]
OR 402.05  ; 精定位气缸B1缩回[M]
ANDLD
ANDNOT 302.06  ; 精定位气缸B1伸出[Pls]
ANDNOT 602.05  ; 精定位气缸B1缩回[A]
ANDNOT 602.06  ; 精定位气缸B1伸出[A]
ANDNOT 802.05  ; 精定位气缸B1原位标志[0002.05]
OUT 402.05  ; 精定位气缸B1缩回[M]
LD TR0
LD 702.06  ; 精定位气缸B1伸出[SW]
OR D1051.05  ; 入钉精定位气缸B1伸出复位
ANDLD
DIFU(013) 302.06  ; 精定位气缸B1伸出[Pls]
LD TR0
LD 302.06  ; 精定位气缸B1伸出[Pls]
OR 402.06  ; 精定位气缸B1伸出[M]
ANDLD
ANDNOT 302.05  ; 精定位气缸B1缩回[Pls]
ANDNOT 602.05  ; 精定位气缸B1缩回[A]
ANDNOT 602.06  ; 精定位气缸B1伸出[A]
ANDNOT 802.06  ; 精定位气缸B1到位标志[0002.06]
OUT 402.06  ; 精定位气缸B1伸出[M]
LD TR0
LD 702.07  ; 精定位气缸B2缩回[SW]
OR D1051.04  ; 入钉精定位气缸B2缩回复位
ANDLD
DIFU(013) 302.07  ; 精定位气缸B2缩回[Pls]
LD TR0
LD 302.07  ; 精定位气缸B2缩回[Pls]
OR 402.07  ; 精定位气缸B2缩回[M]
ANDLD
ANDNOT 302.08  ; 精定位气缸B2伸出[Pls]
ANDNOT 602.07  ; 精定位气缸B2缩回[A]
ANDNOT 602.08  ; 精定位气缸B2伸出[A]
ANDNOT 802.07  ; 精定位气缸B2原位标志[0002.07]
OUT 402.07  ; 精定位气缸B2缩回[M]
LD TR0
LD 702.08  ; 精定位气缸B2伸出[SW]
OR D1051.06  ; 入钉精定位气缸B2伸出复位
ANDLD
DIFU(013) 302.08  ; 精定位气缸B2伸出[Pls]
LD TR0
LD 302.08  ; 精定位气缸B2伸出[Pls]
OR 402.08  ; 精定位气缸B2伸出[M]
ANDLD
ANDNOT 302.07  ; 精定位气缸B2缩回[Pls]
ANDNOT 602.07  ; 精定位气缸B2缩回[A]
ANDNOT 602.08  ; 精定位气缸B2伸出[A]
ANDNOT 802.08  ; 精定位气缸B2到位标志[0002.08]
OUT 402.08  ; 精定位气缸B2伸出[M]

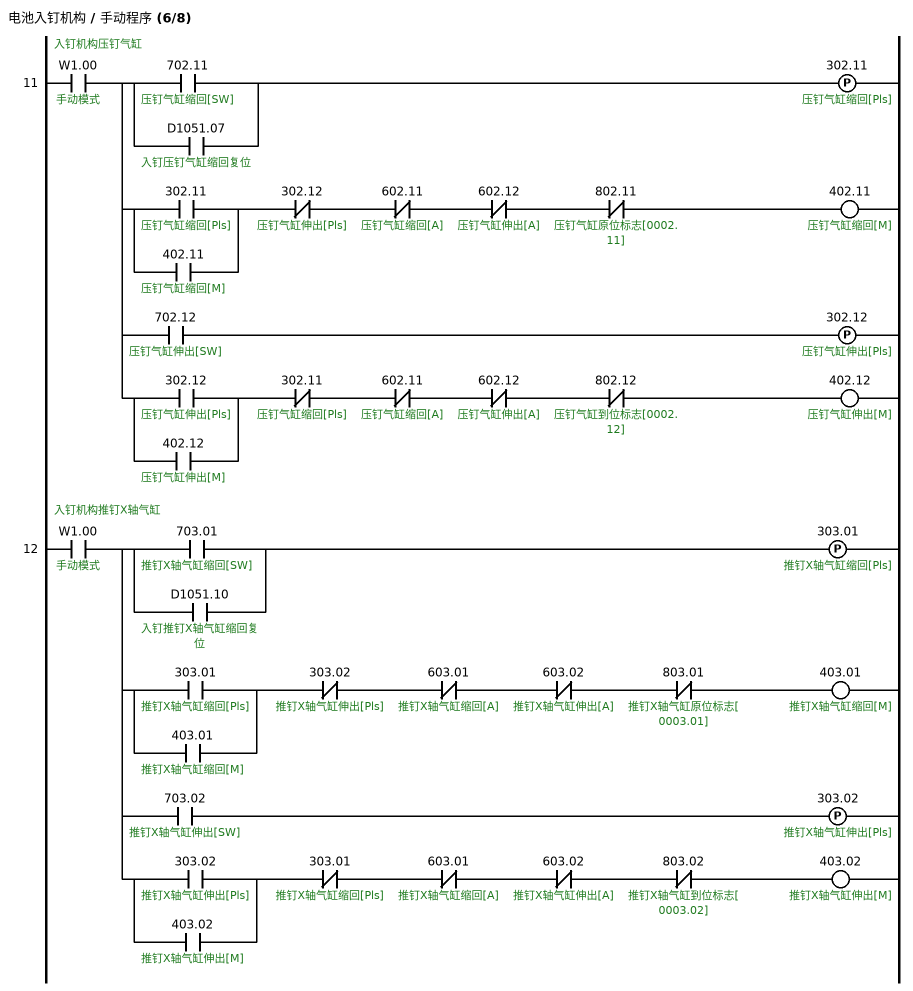
; rung 11: 入钉机构压钉气缸
LD W1.00  ; 手动模式
OUT TR0
LD 702.11  ; 压钉气缸缩回[SW]
OR D1051.07  ; 入钉压钉气缸缩回复位
ANDLD
DIFU(013) 302.11  ; 压钉气缸缩回[Pls]
LD TR0
LD 302.11  ; 压钉气缸缩回[Pls]
OR 402.11  ; 压钉气缸缩回[M]
ANDLD
ANDNOT 302.12  ; 压钉气缸伸出[Pls]
ANDNOT 602.11  ; 压钉气缸缩回[A]
ANDNOT 602.12  ; 压钉气缸伸出[A]
ANDNOT 802.11  ; 压钉气缸原位标志[0002.11]
OUT 402.11  ; 压钉气缸缩回[M]
LD TR0
AND 702.12  ; 压钉气缸伸出[SW]
DIFU(013) 302.12  ; 压钉气缸伸出[Pls]
LD TR0
LD 302.12  ; 压钉气缸伸出[Pls]
OR 402.12  ; 压钉气缸伸出[M]
ANDLD
ANDNOT 302.11  ; 压钉气缸缩回[Pls]
ANDNOT 602.11  ; 压钉气缸缩回[A]
ANDNOT 602.12  ; 压钉气缸伸出[A]
ANDNOT 802.12  ; 压钉气缸到位标志[0002.12]
OUT 402.12  ; 压钉气缸伸出[M]
; rung 12: 入钉机构推钉X轴气缸
LD W1.00  ; 手动模式
OUT TR0
LD 703.01  ; 推钉X轴气缸缩回[SW]
OR D1051.10  ; 入钉推钉X轴气缸缩回复位
ANDLD
DIFU(013) 303.01  ; 推钉X轴气缸缩回[Pls]
LD TR0
LD 303.01  ; 推钉X轴气缸缩回[Pls]
OR 403.01  ; 推钉X轴气缸缩回[M]
ANDLD
ANDNOT 303.02  ; 推钉X轴气缸伸出[Pls]
ANDNOT 603.01  ; 推钉X轴气缸缩回[A]
ANDNOT 603.02  ; 推钉X轴气缸伸出[A]
ANDNOT 803.01  ; 推钉X轴气缸原位标志[0003.01]
OUT 403.01  ; 推钉X轴气缸缩回[M]
LD TR0
AND 703.02  ; 推钉X轴气缸伸出[SW]
DIFU(013) 303.02  ; 推钉X轴气缸伸出[Pls]
LD TR0
LD 303.02  ; 推钉X轴气缸伸出[Pls]
OR 403.02  ; 推钉X轴气缸伸出[M]
ANDLD
ANDNOT 303.01  ; 推钉X轴气缸缩回[Pls]
ANDNOT 603.01  ; 推钉X轴气缸缩回[A]
ANDNOT 603.02  ; 推钉X轴气缸伸出[A]
ANDNOT 803.02  ; 推钉X轴气缸到位标志[0003.02]
OUT 403.02  ; 推钉X轴气缸伸出[M]

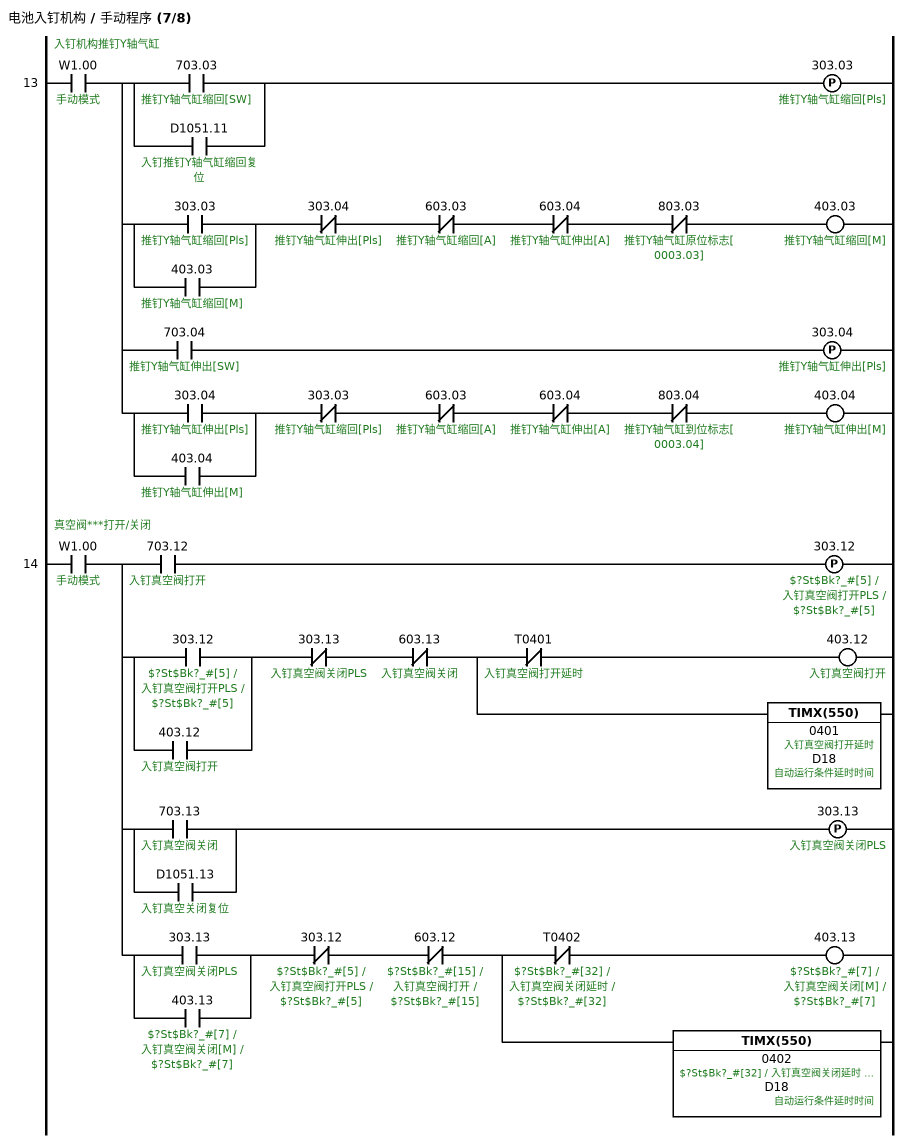
; rung 13: 入钉机构推钉Y轴气缸
LD W1.00  ; 手动模式
OUT TR0
LD 703.03  ; 推钉Y轴气缸缩回[SW]
OR D1051.11  ; 入钉推钉Y轴气缸缩回复位
ANDLD
DIFU(013) 303.03  ; 推钉Y轴气缸缩回[Pls]
LD TR0
LD 303.03  ; 推钉Y轴气缸缩回[Pls]
OR 403.03  ; 推钉Y轴气缸缩回[M]
ANDLD
ANDNOT 303.04  ; 推钉Y轴气缸伸出[Pls]
ANDNOT 603.03  ; 推钉Y轴气缸缩回[A]
ANDNOT 603.04  ; 推钉Y轴气缸伸出[A]
ANDNOT 803.03  ; 推钉Y轴气缸原位标志[0003.03]
OUT 403.03  ; 推钉Y轴气缸缩回[M]
LD TR0
AND 703.04  ; 推钉Y轴气缸伸出[SW]
DIFU(013) 303.04  ; 推钉Y轴气缸伸出[Pls]
LD TR0
LD 303.04  ; 推钉Y轴气缸伸出[Pls]
OR 403.04  ; 推钉Y轴气缸伸出[M]
ANDLD
ANDNOT 303.03  ; 推钉Y轴气缸缩回[Pls]
ANDNOT 603.03  ; 推钉Y轴气缸缩回[A]
ANDNOT 603.04  ; 推钉Y轴气缸伸出[A]
ANDNOT 803.04  ; 推钉Y轴气缸到位标志[0003.04]
OUT 403.04  ; 推钉Y轴气缸伸出[M]
; rung 14: 真空阀***打开/关闭
LD W1.00  ; 手动模式
OUT TR0
AND 703.12  ; 入钉真空阀打开
DIFU(013) 303.12  ; $?St$Bk?_#[5] / 入钉真空阀打开PLS / $?St$Bk?_#[5]
LD TR0
LD 303.12  ; $?St$Bk?_#[5] / 入钉真空阀打开PLS / $?St$Bk?_#[5]
OR 403.12  ; 入钉真空阀打开
ANDLD
ANDNOT 303.13  ; 入钉真空阀关闭PLS
ANDNOT 603.13  ; 入钉真空阀关闭
OUT TR1
ANDNOT T0401  ; 入钉真空阀打开延时
OUT 403.12  ; 入钉真空阀打开
LD TR1
TIMX(550) 0401 D18  ; 自动运行条件延时时间, 入钉真空阀打开延时
LD TR0
LD 703.13  ; 入钉真空阀关闭
OR D1051.13  ; 入钉真空关闭复位
ANDLD
DIFU(013) 303.13  ; 入钉真空阀关闭PLS
LD TR0
LD 303.13  ; 入钉真空阀关闭PLS
OR 403.13  ; $?St$Bk?_#[7] / 入钉真空阀关闭[M] / $?St$Bk?_#[7]
ANDLD
ANDNOT 303.12  ; $?St$Bk?_#[5] / 入钉真空阀打开PLS / $?St$Bk?_#[5]
ANDNOT 603.12  ; $?St$Bk?_#[15] / 入钉真空阀打开 / $?St$Bk?_#[15]
OUT TR0
ANDNOT T0402  ; $?St$Bk?_#[32] / 入钉真空阀关闭延时 / $?St$Bk?_#[32]
OUT 403.13  ; $?St$Bk?_#[7] / 入钉真空阀关闭[M] / $?St$Bk?_#[7]
LD TR0
TIMX(550) 0402 D18  ; 自动运行条件延时时间, $?St$Bk?_#[32] / 入钉真空阀关闭延时 / $?St$Bk?_#[32]

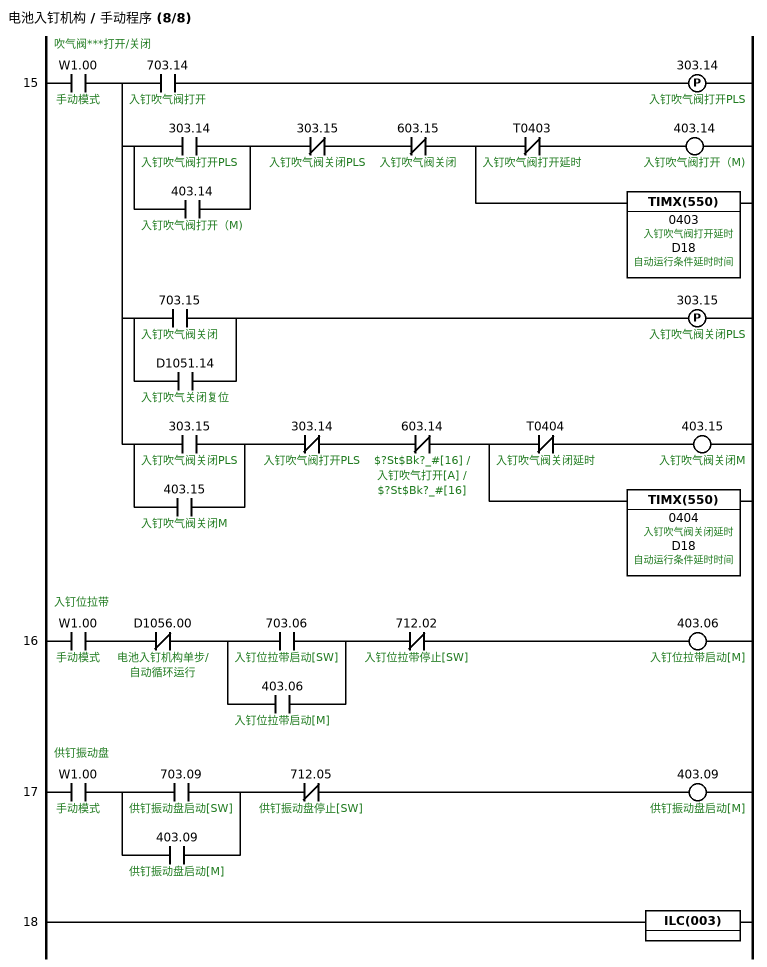
; rung 15: 吹气阀***打开/关闭
LD W1.00  ; 手动模式
OUT TR0
AND 703.14  ; 入钉吹气阀打开
DIFU(013) 303.14  ; 入钉吹气阀打开PLS
LD TR0
LD 303.14  ; 入钉吹气阀打开PLS
OR 403.14  ; 入钉吹气阀打开（M)
ANDLD
ANDNOT 303.15  ; 入钉吹气阀关闭PLS
ANDNOT 603.15  ; 入钉吹气阀关闭
OUT TR1
ANDNOT T0403  ; 入钉吹气阀打开延时
OUT 403.14  ; 入钉吹气阀打开（M)
LD TR1
TIMX(550) 0403 D18  ; 自动运行条件延时时间, 入钉吹气阀打开延时
LD TR0
LD 703.15  ; 入钉吹气阀关闭
OR D1051.14  ; 入钉吹气关闭复位
ANDLD
DIFU(013) 303.15  ; 入钉吹气阀关闭PLS
LD TR0
LD 303.15  ; 入钉吹气阀关闭PLS
OR 403.15  ; 入钉吹气阀关闭M
ANDLD
ANDNOT 303.14  ; 入钉吹气阀打开PLS
ANDNOT 603.14  ; $?St$Bk?_#[16] / 入钉吹气打开[A] / $?St$Bk?_#[16]
OUT TR0
ANDNOT T0404  ; 入钉吹气阀关闭延时
OUT 403.15  ; 入钉吹气阀关闭M
LD TR0
TIMX(550) 0404 D18  ; 自动运行条件延时时间, 入钉吹气阀关闭延时
; rung 16: 入钉位拉带
LD W1.00  ; 手动模式
ANDNOT D1056.00  ; 电池入钉机构单步/自动循环运行
LD 703.06  ; 入钉位拉带启动[SW]
OR 403.06  ; 入钉位拉带启动[M]
ANDLD
ANDNOT 712.02  ; 入钉位拉带停止[SW]
OUT 403.06  ; 入钉位拉带启动[M]
; rung 17: 供钉振动盘
LD W1.00  ; 手动模式
LD 703.09  ; 供钉振动盘启动[SW]
OR 403.09  ; 供钉振动盘启动[M]
ANDLD
ANDNOT 712.05  ; 供钉振动盘停止[SW]
OUT 403.09  ; 供钉振动盘启动[M]
; rung 18
ILC(003)

### Section 自动程序

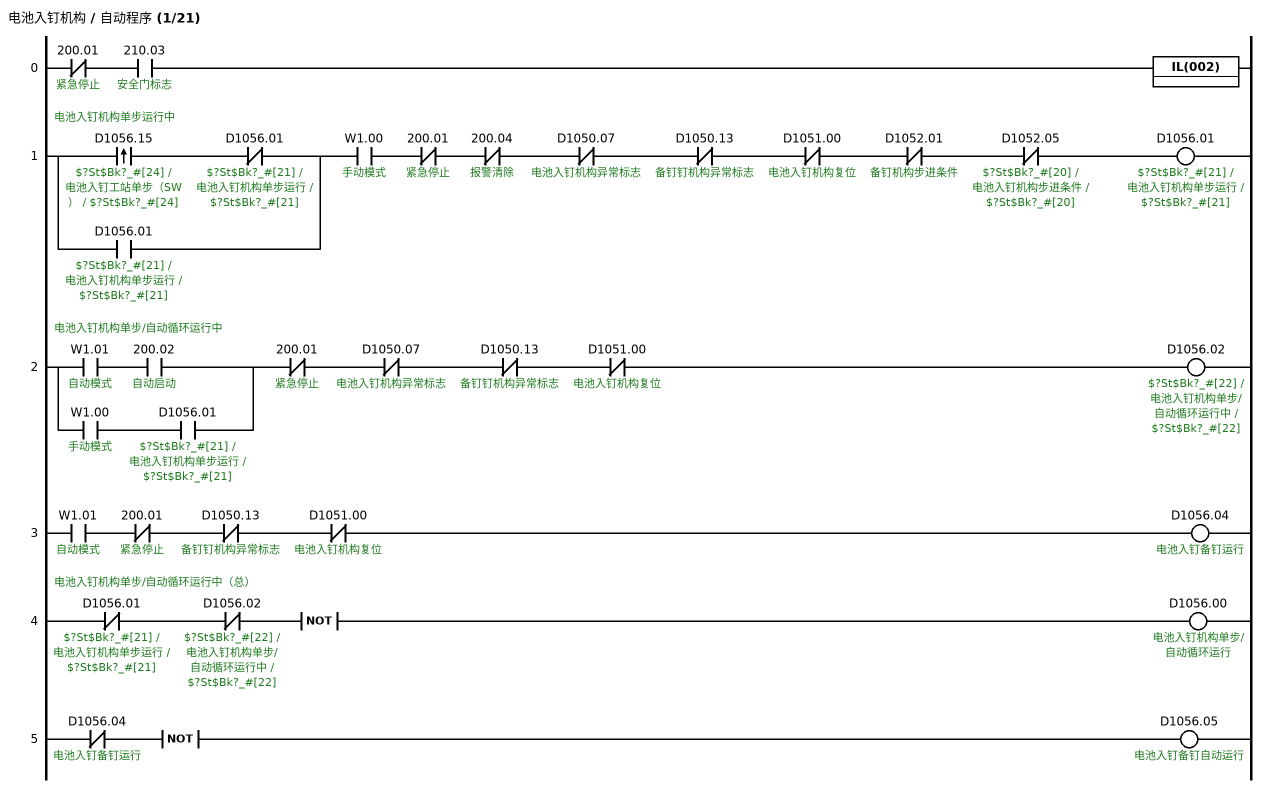
; rung 0
LDNOT 200.01  ; 紧急停止
AND 210.03  ; 安全门标志
IL(002)
; rung 1: 电池入钉机构单步运行中
@LD D1056.15  ; $?St$Bk?_#[24] / 电池入钉工站单步（SW） / $?St$Bk?_#[24]
ANDNOT D1056.01  ; $?St$Bk?_#[21] / 电池入钉机构单步运行 / $?St$Bk?_#[21]
OR D1056.01  ; $?St$Bk?_#[21] / 电池入钉机构单步运行 / $?St$Bk?_#[21]
AND W1.00  ; 手动模式
ANDNOT 200.01  ; 紧急停止
ANDNOT 200.04  ; 报警清除
ANDNOT D1050.07  ; 电池入钉机构异常标志
ANDNOT D1050.13  ; 备钉钉机构异常标志
ANDNOT D1051.00  ; 电池入钉机构复位
ANDNOT D1052.01  ; 备钉机构步进条件
ANDNOT D1052.05  ; $?St$Bk?_#[20] / 电池入钉机构步进条件 / $?St$Bk?_#[20]
OUT D1056.01  ; $?St$Bk?_#[21] / 电池入钉机构单步运行 / $?St$Bk?_#[21]
; rung 2: 电池入钉机构单步/自动循环运行中
LD W1.01  ; 自动模式
AND 200.02  ; 自动启动
LD W1.00  ; 手动模式
AND D1056.01  ; $?St$Bk?_#[21] / 电池入钉机构单步运行 / $?St$Bk?_#[21]
ORLD
ANDNOT 200.01  ; 紧急停止
ANDNOT D1050.07  ; 电池入钉机构异常标志
ANDNOT D1050.13  ; 备钉钉机构异常标志
ANDNOT D1051.00  ; 电池入钉机构复位
OUT D1056.02  ; $?St$Bk?_#[22] / 电池入钉机构单步/自动循环运行中 / $?St$Bk?_#[22]
; rung 3
LD W1.01  ; 自动模式
ANDNOT 200.01  ; 紧急停止
ANDNOT D1050.13  ; 备钉钉机构异常标志
ANDNOT D1051.00  ; 电池入钉机构复位
OUT D1056.04  ; 电池入钉备钉运行
; rung 4: 电池入钉机构单步/自动循环运行中（总）
LDNOT D1056.01  ; $?St$Bk?_#[21] / 电池入钉机构单步运行 / $?St$Bk?_#[21]
ANDNOT D1056.02  ; $?St$Bk?_#[22] / 电池入钉机构单步/自动循环运行中 / $?St$Bk?_#[22]
NOT(520)
OUT D1056.00  ; 电池入钉机构单步/自动循环运行
; rung 5
LDNOT D1056.04  ; 电池入钉备钉运行
NOT(520)
OUT D1056.05  ; 电池入钉备钉自动运行

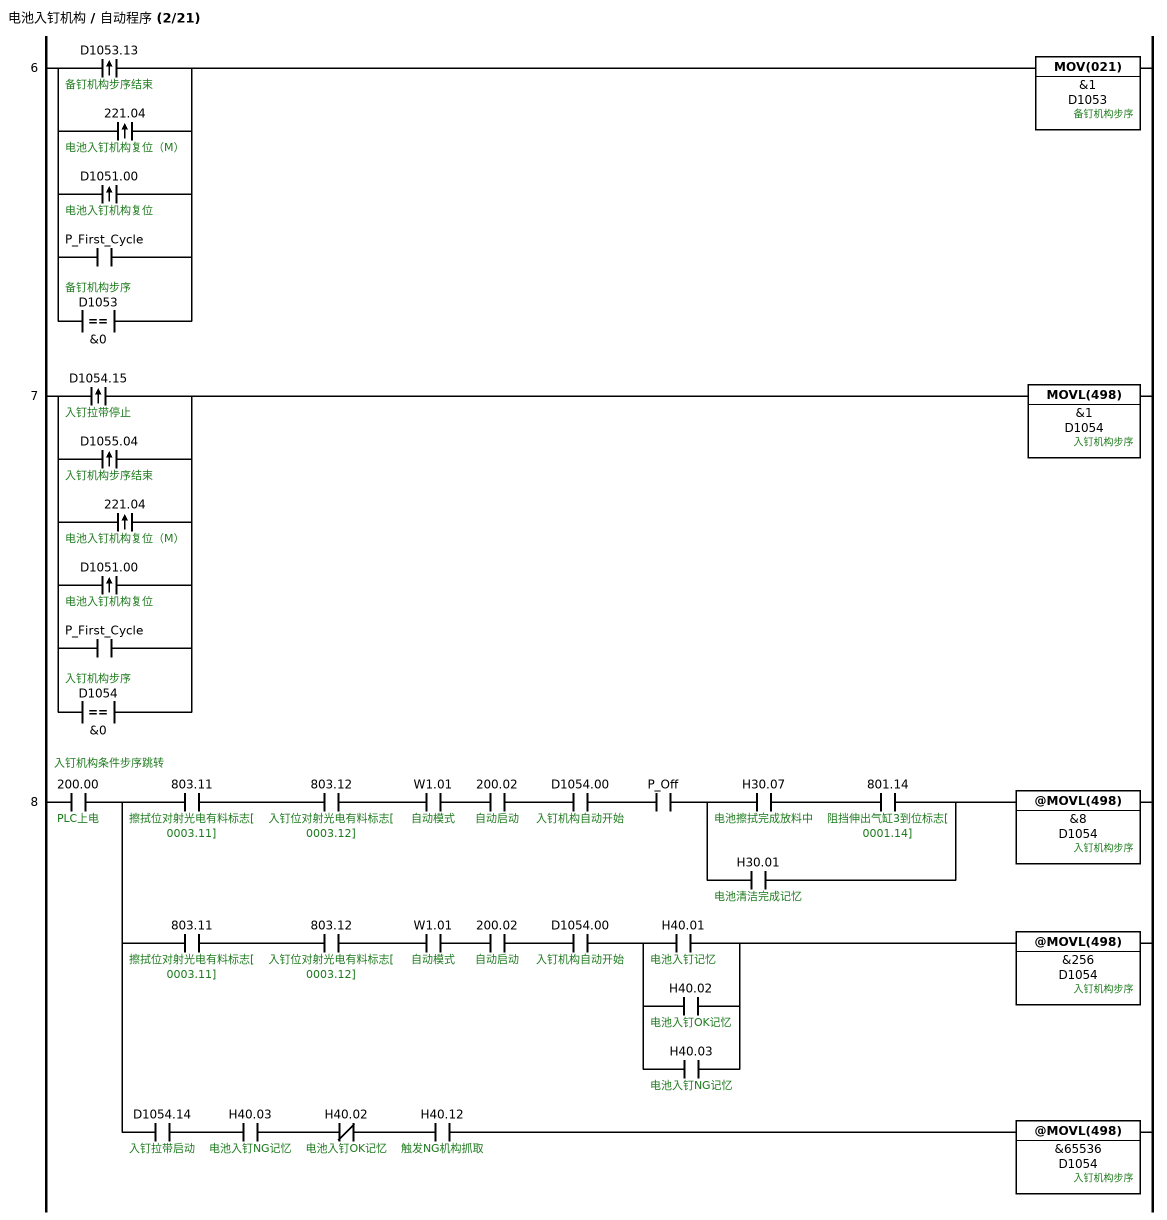
; rung 6
@LD D1053.13  ; 备钉机构步序结束
@OR 221.04  ; 电池入钉机构复位（M）
@OR D1051.00  ; 电池入钉机构复位
OR P_First_Cycle
OR=(300) D1053 &0  ; 备钉机构步序
MOV(021) &1 D1053  ; 备钉机构步序
; rung 7
@LD D1054.15  ; 入钉拉带停止
@OR D1055.04  ; 入钉机构步序结束
@OR 221.04  ; 电池入钉机构复位（M）
@OR D1051.00  ; 电池入钉机构复位
OR P_First_Cycle
OR=L(301) D1054 &0  ; 入钉机构步序
MOVL(498) &1 D1054  ; 入钉机构步序
; rung 8: 入钉机构条件步序跳转
LD 200.00  ; PLC上电
OUT TR0
AND 803.11  ; 擦拭位对射光电有料标志[0003.11]
AND 803.12  ; 入钉位对射光电有料标志[0003.12]
AND W1.01  ; 自动模式
AND 200.02  ; 自动启动
AND D1054.00  ; 入钉机构自动开始
AND P_Off
LD H30.07  ; 电池擦拭完成放料中
AND 801.14  ; 阻挡伸出气缸3到位标志[0001.14]
OR H30.01  ; 电池清洁完成记忆
ANDLD
@MOVL(498) &8 D1054  ; 入钉机构步序
LD TR0
AND 803.11  ; 擦拭位对射光电有料标志[0003.11]
AND 803.12  ; 入钉位对射光电有料标志[0003.12]
AND W1.01  ; 自动模式
AND 200.02  ; 自动启动
AND D1054.00  ; 入钉机构自动开始
LD H40.01  ; 电池入钉记忆
OR H40.02  ; 电池入钉OK记忆
OR H40.03  ; 电池入钉NG记忆
ANDLD
@MOVL(498) &256 D1054  ; 入钉机构步序
LD TR0
AND D1054.14  ; 入钉拉带启动
AND H40.03  ; 电池入钉NG记忆
ANDNOT H40.02  ; 电池入钉OK记忆
AND H40.12  ; 触发NG机构抓取
@MOVL(498) &65536 D1054  ; 入钉机构步序

